(* PLC project mtcs_m2, Institute of Astronomy Onto 0.0.1 *)
(* stored: creationDateTime 2025-03-28T22:57:03.477723, modificationDateTime 2025-03-28T22:57:03.477723 *)

TYPE M2Axes : (X := 0, Y := 1, Z := 2, TILTX := 3, TILTY := 4);
END_TYPE

TYPE M2MoveProcedureStates : (IDLE := 0, ABORTED := 1, PREPARE_PROCESS := 2, MOVING := 3, MOVING_TO_ANTI_BACKLASH_POSITION := 4, MOVING_CLOSE_TO_FINAL_POSITION := 5, MOVING_TO_FINAL_POSITION := 6, ERROR := 7, ABORTING := 8);
END_TYPE

TYPE M2Parts : STRUCT
  {attribute 'TcHmiSymbol.Show'}
  powerRelay : SimpleRelay;  (* Relay to power on/off the power of the M2 field electricity *)
  {attribute 'TcHmiSymbol.Show'}
  heater : SimpleRelay;  (* Digital output to power on/off the heater of M2 *)
  {attribute 'TcHmiSymbol.Show'}
  x : M2XAxis;  (* The X axis *)
  {attribute 'TcHmiSymbol.Show'}
  y : M2YAxis;  (* The Y axis *)
  {attribute 'TcHmiSymbol.Show'}
  z : M2ZAxis;  (* The Z axis *)
  {attribute 'TcHmiSymbol.Show'}
  tiltX : M2TiltXAxis;  (* The TiltX axis *)
  {attribute 'TcHmiSymbol.Show'}
  tiltY : M2TiltYAxis;  (* The TiltY axis *)
  {attribute 'TcHmiSymbol.Show'}
  multiplexer : M2Multiplexer;  (* The multiplexer inputs and outputs *)
  {attribute 'TcHmiSymbol.Show'}
  configManager : ConfigManager;  (* The config manager (to load/save/activate configuration data) *)
  {attribute 'TcHmiSymbol.Show'}
  moveStepsProcedure : M2MoveStepsProcedure;  (* The move steps procedure *)
  {attribute 'TcHmiSymbol.Show'}
  movePositionProcedure : M2MovePositionProcedure;  (* The move to a certain position procedure *)
END_STRUCT;
END_TYPE

TYPE M2MultiplexerParts : STRUCT
  {attribute 'TcHmiSymbol.Show'}
  A : SimpleRelay;  (* Output A of the multiplexer corresponding with the selected axis *)
  {attribute 'TcHmiSymbol.Show'}
  B : SimpleRelay;  (* Output B of the multiplexer corresponding with the selected axis *)
  {attribute 'TcHmiSymbol.Show'}
  C : SimpleRelay;  (* Output C of the multiplexer corresponding with the selected axis *)
  {attribute 'TcHmiSymbol.Show'}
  driveEnable : SimpleRelay;  (* Enabled (TRUE) if the drive selected by the multiplexer must be enabled, Disabled (FALSE) if it must be disabled *)
  {attribute 'TcHmiSymbol.Show'}
  CW : SimpleRelay;  (* Enabled (TRUE) if the motor selected by the multiplexer will run in CW direction (- motion on the screw), Disabled (FALSE) if it will run in CCW direction (+ motion on the screw) *)
  {attribute 'TcHmiSymbol.Show'}
  release : SimpleRelay;  (* Disabled (FALSE) if the motor selected by the multiplexer must be braking, Enabled (TRUE) if it must be released *)
END_STRUCT;
END_TYPE

TYPE M2ZAxisParts : STRUCT
  {attribute 'TcHmiSymbol.Show'}
  highSpeed : SimpleRelay;  (* Enabled (TRUE) to enable the high-speed motion of the Z axis, Disabled (FALSE) to leave it low-speed *)
  {attribute 'TcHmiSymbol.Show'}
  encoder : SSIEncoder;  (* The SSI encoder of the Z axis *)
END_STRUCT;
END_TYPE

TYPE M2Processes : STRUCT
  {attribute 'TcHmiSymbol.Show'}
  initialize : Process;  (* Start initializing *)
  {attribute 'TcHmiSymbol.Show'}
  lock : Process;  (* Lock the system *)
  {attribute 'TcHmiSymbol.Show'}
  unlock : Process;  (* Unlock the system *)
  {attribute 'TcHmiSymbol.Show'}
  changeOperatingState : ChangeOperatingStateProcess;  (* Change the operating state (e.g. AUTO, MANUAL, ...) *)
  {attribute 'TcHmiSymbol.Show'}
  moveAbsolute : M2MoveProcess;  (* Move the position of one axis in an absolute way *)
  {attribute 'TcHmiSymbol.Show'}
  moveRelative : M2MoveProcess;  (* Move the position of one axis relative to the current position *)
  {attribute 'TcHmiSymbol.Show'}
  moveSteps : M2MoveStepsProcess;  (* Move the position of one axis by providing a number of steps (i.e. motor pulses) *)
  {attribute 'TcHmiSymbol.Show'}
  doThermalFocus : Process;  (* Do a thermal focus for the currently active focus *)
  {attribute 'TcHmiSymbol.Show'}
  doThermalFocusForStationName : M2DoThermalFocusForStationName;  (* Do a thermal focus for a specified focal station (based on the configured name of the station) *)
  {attribute 'TcHmiSymbol.Show'}
  doThermalFocusForStationPosition : M2DoThermalFocusForStationPosition;  (* Do a thermal focus for a specified focal station (based on the station numerical ID) *)
  {attribute 'TcHmiSymbol.Show'}
  verifyFixedPositions : Process;  (* Verify (and adjust if necessary) the fixed positions of X, Y, TiltX, and TiltY *)
  {attribute 'TcHmiSymbol.Show'}
  powerOn : Process;  (* Power on the M2 electricity *)
  {attribute 'TcHmiSymbol.Show'}
  powerOff : Process;  (* Power off the M2 electricity *)
  {attribute 'TcHmiSymbol.Show'}
  abort : Process;  (* Abort the move procedure *)
END_STRUCT;
END_TYPE

TYPE M2MultiplexerProcesses : STRUCT
  {attribute 'TcHmiSymbol.Show'}
  selectAxis : M2SelectAxisProcess;  (* Select an axis *)
END_STRUCT;
END_TYPE

TYPE M2Statuses : STRUCT
  {attribute 'TcHmiSymbol.Show'}
  initializationStatus : InitializationStatus;
  {attribute 'TcHmiSymbol.Show'}
  poweredStatus : PoweredStatus;
  {attribute 'TcHmiSymbol.Show'}
  healthStatus : HealthStatus;
  {attribute 'TcHmiSymbol.Show'}
  busyStatus : BusyStatus;
  {attribute 'TcHmiSymbol.Show'}
  operatingStatus : OperatingStatus;
END_STRUCT;
END_TYPE

TYPE M2MultiplexerStatuses : STRUCT
  {attribute 'TcHmiSymbol.Show'}
  healthStatus : HealthStatus;  (* Is the selected drive healthy? *)
  {attribute 'TcHmiSymbol.Show'}
  busyStatus : BusyStatus;  (* Is the selected drive busy? *)
END_STRUCT;
END_TYPE

TYPE M2XAxisStatuses : STRUCT
  {attribute 'TcHmiSymbol.Show'}
  healthStatus : HealthStatus;  (* Is the axis healthy? *)
END_STRUCT;
END_TYPE

TYPE M2YAxisStatuses : STRUCT
  {attribute 'TcHmiSymbol.Show'}
  healthStatus : HealthStatus;  (* Is the axis healthy? *)
END_STRUCT;
END_TYPE

TYPE M2TiltXAxisStatuses : STRUCT
  {attribute 'TcHmiSymbol.Show'}
  healthStatus : HealthStatus;  (* Is the axis healthy? *)
END_STRUCT;
END_TYPE

TYPE M2TiltYAxisStatuses : STRUCT
  {attribute 'TcHmiSymbol.Show'}
  healthStatus : HealthStatus;  (* Is the axis healthy? *)
END_STRUCT;
END_TYPE

TYPE M2ZAxisStatuses : STRUCT
  {attribute 'TcHmiSymbol.Show'}
  healthStatus : HealthStatus;  (* Is the axis healthy? *)
END_STRUCT;
END_TYPE

TYPE M2MoveStepsProcedureStatuses : STRUCT
  {attribute 'TcHmiSymbol.Show'}
  busyStatus : BusyStatus;  (* Is the M2MoveStepsProcedure in a busy state? *)
  {attribute 'TcHmiSymbol.Show'}
  healthStatus : HealthStatus;  (* Is the M2MoveStepsProcedure in a healthy state? *)
END_STRUCT;
END_TYPE

TYPE M2MovePositionProcedureStatuses : STRUCT
  {attribute 'TcHmiSymbol.Show'}
  busyStatus : BusyStatus;  (* Is the M2MoveAbsoluteProcedure in a busy state? *)
  {attribute 'TcHmiSymbol.Show'}
  healthStatus : HealthStatus;  (* Is the M2MoveAbsoluteProcedure in a healthy state? *)
END_STRUCT;
END_TYPE

TYPE M2Config : STRUCT
  {attribute 'TcHmiSymbol.Show'}
  x : M2PotentiometerAxisConfig;  (* The config of the X axis *)
  {attribute 'TcHmiSymbol.Show'}
  y : M2PotentiometerAxisConfig;  (* The config of the Y axis *)
  {attribute 'TcHmiSymbol.Show'}
  z : M2ZAxisConfig;  (* The config of the Z axis *)
  {attribute 'TcHmiSymbol.Show'}
  tiltX : M2PotentiometerAxisConfig;  (* The config of the tiltX axis *)
  {attribute 'TcHmiSymbol.Show'}
  tiltY : M2PotentiometerAxisConfig;  (* The config of the tiltY axis *)
  {attribute 'TcHmiSymbol.Show'}
  thermalFocus : M2ThermalFocusConfig;  (* The thermal focus coefficients for all focal stations *)
  {attribute 'TcHmiSymbol.Show'}
  waitAfterPowerOn : LREAL;  (* Time (in seconds) to wait after the field electricity of M2 have been powered on *)
  {attribute 'TcHmiSymbol.Show'}
  waitAfterPowerOff : LREAL;  (* Time (in seconds) to wait after the field electricity of M2 have been powered off *)
  {attribute 'TcHmiSymbol.Show'}
  powerOffTimeout : LREAL;  (* If no new command is sent to M2 within this time (in seconds) after completion of the last command, M2 will be powered off automatically *)
  {attribute 'TcHmiSymbol.Show'}
  fixedXPosition : LREAL;  (* The fixed X position in mm *)
  {attribute 'TcHmiSymbol.Show'}
  fixedXPositionTolerance : LREAL;  (* If the X position is within fixedXPosition +/- this tolerance, there's no need to adjust it *)
  {attribute 'TcHmiSymbol.Show'}
  fixedYPosition : LREAL;  (* The fixed Y position in mm *)
  {attribute 'TcHmiSymbol.Show'}
  fixedYPositionTolerance : LREAL;  (* If the Y position is within fixedYPosition +/- this tolerance, there's no need to adjust it *)
  {attribute 'TcHmiSymbol.Show'}
  fixedTiltXPosition : LREAL;  (* The fixed TiltX position in mm *)
  {attribute 'TcHmiSymbol.Show'}
  fixedTiltXPositionTolerance : LREAL;  (* If the TiltX position is within fixedTiltXPosition +/- this tolerance, there's no need to adjust it *)
  {attribute 'TcHmiSymbol.Show'}
  fixedTiltYPosition : LREAL;  (* The fixed TiltY position in mm *)
  {attribute 'TcHmiSymbol.Show'}
  fixedTiltYPositionTolerance : LREAL;  (* If the TiltY position is within fixedTiltYPosition +/- this tolerance, there's no need to adjust it *)
  {attribute 'TcHmiSymbol.Show'}
  verifyFixedPositinsOnThermalFocus : BOOL;  (* Each time a theremal focus is done, verify the fixed positions (and adjust them if they fall out of the tolerance) *)
END_STRUCT;
END_TYPE

TYPE M2ThermalFocusStationConfig : STRUCT
  {attribute 'TcHmiSymbol.Show'}
  offset : LREAL;  (* focus = offset + topCoefficient*topTemperature + centreCoefficient*centreTemperature + mirrorCellCoefficient*mirrorCellTemperature *)
  {attribute 'TcHmiSymbol.Show'}
  topCoefficient : LREAL;  (* focus = offset + topCoefficient*topTemperature + centreCoefficient*centreTemperature + mirrorCellCoefficient*mirrorCellTemperature *)
  {attribute 'TcHmiSymbol.Show'}
  centreCoefficient : LREAL;  (* focus = offset + topCoefficient*topTemperature + centreCoefficient*centreTemperature + mirrorCellCoefficient*mirrorCellTemperature *)
  {attribute 'TcHmiSymbol.Show'}
  mirrorCellCoefficient : LREAL;  (* focus = offset + topCoefficient*topTemperature + centreCoefficient*centreTemperature + mirrorCellCoefficient*mirrorCellTemperature *)
END_STRUCT;
END_TYPE

TYPE M2ThermalFocusConfig : STRUCT
  {attribute 'TcHmiSymbol.Show'}
  cassegrain : M2ThermalFocusStationConfig;  (* Cassegrain thermal focus config *)
  {attribute 'TcHmiSymbol.Show'}
  nasmythA : M2ThermalFocusStationConfig;  (* Nasmyth A thermal focus config *)
  {attribute 'TcHmiSymbol.Show'}
  nasmythB : M2ThermalFocusStationConfig;  (* Nasmyth B thermal focus config *)
  {attribute 'TcHmiSymbol.Show'}
  nasmythC : M2ThermalFocusStationConfig;  (* Nasmyth C thermal focus config *)
  {attribute 'TcHmiSymbol.Show'}
  nasmythD : M2ThermalFocusStationConfig;  (* Nasmyth D thermal focus config *)
  {attribute 'TcHmiSymbol.Show'}
  other0 : M2ThermalFocusStationConfig;  (* Other 0 thermal focus config *)
  {attribute 'TcHmiSymbol.Show'}
  other1 : M2ThermalFocusStationConfig;  (* Other 1 thermal focus config *)
  {attribute 'TcHmiSymbol.Show'}
  other2 : M2ThermalFocusStationConfig;  (* Other 2 thermal focus config *)
  {attribute 'TcHmiSymbol.Show'}
  other3 : M2ThermalFocusStationConfig;  (* Other 3 thermal focus config *)
  {attribute 'TcHmiSymbol.Show'}
  other4 : M2ThermalFocusStationConfig;  (* Other 4 thermal focus config *)
END_STRUCT;
END_TYPE

TYPE M2AxisGeneralConfig : STRUCT
  {attribute 'TcHmiSymbol.Show'}
  measurement : MeasurementConfig;  (* Configure the position measurement *)
  {attribute 'TcHmiSymbol.Show'}
  stoppingSteps : UDINT;  (* The number of steps to be expected between the time at which the PLC realizes that the brake release signal must be set, and the time that the axis is fully stopped (for Z axis: at low speed) *)
  {attribute 'TcHmiSymbol.Show'}
  finalSenseCW : BOOL;  (* TRUE if the motor final sense must be ClockWise (- motion on the screw), FALSE if the motor final sense must be CounterClockWise (+ motion on the screw) (for Z axis: at low speed) *)
  {attribute 'TcHmiSymbol.Show'}
  closePosition : UDINT;  (* The number of steps between the Close position (C) and final position (F) *)
  {attribute 'TcHmiSymbol.Show'}
  antiBacklashPosition : UDINT;  (* The number of steps between the Anti-backlash position (A) and final position (F) *)
  {attribute 'TcHmiSymbol.Show'}
  waitAfterMove : LREAL;  (* Time (in seconds) to wait after the axis has been moved *)
  {attribute 'TcHmiSymbol.Show'}
  timeout : LREAL;  (* Timeout for a movement, in seconds (for Z-axis: at low speed) *)
  {attribute 'TcHmiSymbol.Show'}
  verifyPositionOnInitialization : BOOL;  (* Verify the fixed positions (and adjust them if they fall out of the tolerance) during the Initialization procedure *)
END_STRUCT;
END_TYPE

TYPE M2ZAxisConfig : STRUCT
  {attribute 'TcHmiSymbol.Show'}
  general : M2AxisGeneralConfig;  (* Settings which are general for all axes *)
  {attribute 'TcHmiSymbol.Show'}
  highSpeedStoppingSteps : UDINT;  (* The number of steps to be expected between the time at which the PLC realizes that the brake release signal must be set, and the time that the axis is fully stopped at high speed *)
  {attribute 'TcHmiSymbol.Show'}
  highSpeedTimeout : LREAL;  (* Timeout for a fast movement of the Z axis (in seconds) *)
END_STRUCT;
END_TYPE

TYPE M2PotentiometerAxisConfig : STRUCT
  {attribute 'TcHmiSymbol.Show'}
  general : M2AxisGeneralConfig;  (* Settings which are general for all axes *)
  {attribute 'TcHmiSymbol.Show'}
  voltageCorrectionFactor : LREAL;  (* Position = voltage * correctionFactor * voltageToPosition *)
END_STRUCT;
END_TYPE

TYPE M2ConstantsZ : STRUCT
  {attribute 'TcHmiSymbol.Show'}
  MOT_TO_RED_RATIO : LREAL := 134.0;  (* Motor reduction ratio *)
  {attribute 'TcHmiSymbol.Show'}
  RED_TO_SCREW_RATIO : LREAL := 2.0;  (* Transmission ratio between the motor reduction and the screw *)
  {attribute 'TcHmiSymbol.Show'}
  SCREW_TO_ENC_RATIO : LREAL := 1.0;  (* Transmission ratio between the encoder and the screw *)
  {attribute 'TcHmiSymbol.Show'}
  MIN_POSITION : LREAL := 0.0;  (* Minimum position of the axis, in micrometer *)
  {attribute 'TcHmiSymbol.Show'}
  MAX_POSITION : LREAL := 50000.0;  (* Maximum position of the axis, in micrometer *)
  {attribute 'TcHmiSymbol.Show'}
  SCREW_PITCH : LREAL := 2000.0;  (* Screw pitch, in micrometer *)
  {attribute 'TcHmiSymbol.Show'}
  FEEDBACK_RESOLUTION : LREAL := 32.0;  (* Motor feedback resolution (pulses per revolution of the motor rotor) *)
END_STRUCT;
END_TYPE

TYPE M2ConstantsX : STRUCT
  {attribute 'TcHmiSymbol.Show'}
  MOT_TO_RED_RATIO : LREAL := 415.0;  (* Motor reduction ratio *)
  {attribute 'TcHmiSymbol.Show'}
  RED_TO_SCREW_RATIO : LREAL := 2.0;  (* Transmission ratio between the motor reduction and the screw *)
  {attribute 'TcHmiSymbol.Show'}
  SCREW_TO_POT_RATIO : LREAL := 0.5;  (* Transmission ratio between the potentiometer and the screw *)
  {attribute 'TcHmiSymbol.Show'}
  MIN_POSITION : LREAL := 400.0;  (* Minimum position of the axis, in micrometer *)
  {attribute 'TcHmiSymbol.Show'}
  MAX_POSITION : LREAL := 4700.0;  (* Maximum position of the axis, in micrometer *)
  {attribute 'TcHmiSymbol.Show'}
  SCREW_PITCH : LREAL := 1000.0;  (* Screw pitch, in micrometer *)
  {attribute 'TcHmiSymbol.Show'}
  FEEDBACK_RESOLUTION : LREAL := 3.0;  (* Motor feedback resolution (pulses per revolution of the motor rotor) *)
  {attribute 'TcHmiSymbol.Show'}
  POTENTIOMETER_REVOLUTIONS : LREAL := 10.0;  (* Max number of revolutions of the potentiometer *)
END_STRUCT;
END_TYPE

TYPE M2ConstantsY : STRUCT
  {attribute 'TcHmiSymbol.Show'}
  MOT_TO_RED_RATIO : LREAL := 415.0;  (* Motor reduction ratio *)
  {attribute 'TcHmiSymbol.Show'}
  RED_TO_SCREW_RATIO : LREAL := 2.0;  (* Transmission ratio between the motor reduction and the screw *)
  {attribute 'TcHmiSymbol.Show'}
  SCREW_TO_POT_RATIO : LREAL := 0.5;  (* Transmission ratio between the potentiometer and the screw *)
  {attribute 'TcHmiSymbol.Show'}
  MIN_POSITION : LREAL := 400.0;  (* Minimum position of the axis, in micrometer *)
  {attribute 'TcHmiSymbol.Show'}
  MAX_POSITION : LREAL := 4700.0;  (* Maximum position of the axis, in micrometer *)
  {attribute 'TcHmiSymbol.Show'}
  SCREW_PITCH : LREAL := 1000.0;  (* Screw pitch, in micrometer *)
  {attribute 'TcHmiSymbol.Show'}
  FEEDBACK_RESOLUTION : LREAL := 3.0;  (* Motor feedback resolution (pulses per revolution of the motor rotor) *)
  {attribute 'TcHmiSymbol.Show'}
  POTENTIOMETER_REVOLUTIONS : LREAL := 10.0;  (* Max number of revolutions of the potentiometer *)
END_STRUCT;
END_TYPE

TYPE M2ConstantsTiltX : STRUCT
  {attribute 'TcHmiSymbol.Show'}
  MOT_TO_RED_RATIO : LREAL := 1526.0;  (* Motor reduction ratio *)
  {attribute 'TcHmiSymbol.Show'}
  RED_TO_SCREW_RATIO : LREAL := 2.0;  (* Transmission ratio between the motor reduction and the screw *)
  {attribute 'TcHmiSymbol.Show'}
  SCREW_TO_POT_RATIO : LREAL := 0.5;  (* Transmission ratio between the potentiometer and the screw *)
  {attribute 'TcHmiSymbol.Show'}
  MIN_POSITION : LREAL := 260.0;  (* Minimum position of the axis, in micrometer *)
  {attribute 'TcHmiSymbol.Show'}
  MAX_POSITION : LREAL := 1200.0;  (* Maximum position of the axis, in micrometer *)
  {attribute 'TcHmiSymbol.Show'}
  SCREW_PITCH : LREAL := 1000.0;  (* Screw pitch, in micrometer *)
  {attribute 'TcHmiSymbol.Show'}
  FEEDBACK_RESOLUTION : LREAL := 3.0;  (* Motor feedback resolution (pulses per revolution of the motor rotor) *)
  {attribute 'TcHmiSymbol.Show'}
  POTENTIOMETER_REVOLUTIONS : LREAL := 3.0;  (* Max number of revolutions of the potentiometer *)
END_STRUCT;
END_TYPE

TYPE M2ConstantsTiltY : STRUCT
  {attribute 'TcHmiSymbol.Show'}
  MOT_TO_RED_RATIO : LREAL := 1526.0;  (* Motor reduction ratio *)
  {attribute 'TcHmiSymbol.Show'}
  RED_TO_SCREW_RATIO : LREAL := 2.0;  (* Transmission ratio between the motor reduction and the screw *)
  {attribute 'TcHmiSymbol.Show'}
  SCREW_TO_POT_RATIO : LREAL := 0.5;  (* Transmission ratio between the potentiometer and the screw *)
  {attribute 'TcHmiSymbol.Show'}
  MIN_POSITION : LREAL := 180.0;  (* Minimum position of the axis, in micrometer *)
  {attribute 'TcHmiSymbol.Show'}
  MAX_POSITION : LREAL := 1200.0;  (* Maximum position of the axis, in micrometer *)
  {attribute 'TcHmiSymbol.Show'}
  SCREW_PITCH : LREAL := 1000.0;  (* Screw pitch, in micrometer *)
  {attribute 'TcHmiSymbol.Show'}
  FEEDBACK_RESOLUTION : LREAL := 3.0;  (* Motor feedback resolution (pulses per revolution of the motor rotor) *)
  {attribute 'TcHmiSymbol.Show'}
  POTENTIOMETER_REVOLUTIONS : LREAL := 3.0;  (* Max number of revolutions of the potentiometer *)
END_STRUCT;
END_TYPE

TYPE M2SelectAxisProcessArgs : STRUCT
  {attribute 'TcHmiSymbol.Show'}
  axis : M2Axes;  (* The axis to select *)
END_STRUCT;
END_TYPE

TYPE M2MoveProcessArgs : STRUCT
  {attribute 'TcHmiSymbol.Show'}
  axis : M2Axes;  (* The axis to move *)
  {attribute 'TcHmiSymbol.Show'}
  position : LREAL;  (* Move to a certain position in millimeters *)
END_STRUCT;
END_TYPE

TYPE M2MoveStepsProcessArgs : STRUCT
  {attribute 'TcHmiSymbol.Show'}
  axis : M2Axes;  (* The axis to move *)
  {attribute 'TcHmiSymbol.Show'}
  steps : UDINT;  (* Move a certain number of steps *)
  {attribute 'TcHmiSymbol.Show'}
  cw : BOOL;  (* True if the axis should be moved in CW (negative) direction *)
  {attribute 'TcHmiSymbol.Show'}
  fast : BOOL;  (* True if the axis should be moved fast (only used in case of Z-axis!) *)
END_STRUCT;
END_TYPE

TYPE M2DoThermalFocusForStationPositionArgs : STRUCT
  {attribute 'TcHmiSymbol.Show'}
  station : M3PositionIDs;  (* The station numerical ID for which the thermal focus should be executed *)
END_STRUCT;
END_TYPE

TYPE M2DoThermalFocusForStationNameArgs : STRUCT
  {attribute 'TcHmiSymbol.Show'}
  station : STRING;  (* The configured station name, for which the thermal focus should be executed *)
END_STRUCT;
END_TYPE

FUNCTION_BLOCK SM_M2
  VAR_INPUT
    {attribute 'TcHmiSymbol.Show'}
    {attribute 'OPC.UA.DA' := '1'}
    {attribute 'OPC.UA.DA.Access' := '1'}
    editableConfig : M2Config;  (* Editable configuration of the M2 subsystem *)
  END_VAR
  VAR_OUTPUT
    {attribute 'OPC.UA.DA' := '1'}
    {attribute 'OPC.UA.DA.Access' := '1'}
    {attribute 'TcHmiSymbol.Show'}
    actualStatus : STRING;  (* Current status description *)
    {attribute 'TcHmiSymbol.Show'}
    previousStatus : STRING;  (* Previous status description *)
    {attribute 'TcHmiSymbol.Show'}
    {attribute 'OPC.UA.DA' := '1'}
    {attribute 'OPC.UA.DA.Access' := '1'}
    config : M2Config;  (* Active configuration of the M2 subsystem *)
    {attribute 'TcHmiSymbol.Show'}
    {attribute 'OPC.UA.DA' := '1'}
    {attribute 'OPC.UA.DA.Access' := '1'}
    selectedAxis : M2Axes;  (* The axis which is currently selected by the multiplexer *)
    {attribute 'TcHmiSymbol.Show'}
    {attribute 'OPC.UA.DA' := '1'}
    {attribute 'OPC.UA.DA.Access' := '1'}
    selectedAxisName : STRING;  (* The name of the axis which is currently selected by the multiplexer *)
    {attribute 'TcHmiSymbol.Show'}
    {attribute 'OPC.UA.DA' := '1'}
    {attribute 'OPC.UA.DA.Access' := '1'}
    powerOffTimer : LREAL;  (* Number of seconds before the power of the M2 field electricity will be powered off automatically *)
    {attribute 'TcHmiSymbol.Show'}
    {attribute 'OPC.UA.DA' := '1'}
    {attribute 'OPC.UA.DA.Access' := '1'}
    thermalFocusCassegrain : LinearPosition;  (* Thermal focus position for cassegrain *)
    {attribute 'TcHmiSymbol.Show'}
    {attribute 'OPC.UA.DA' := '1'}
    {attribute 'OPC.UA.DA.Access' := '1'}
    thermalFocusNasmythA : LinearPosition;  (* Thermal focus position for nasmyth A *)
    {attribute 'TcHmiSymbol.Show'}
    {attribute 'OPC.UA.DA' := '1'}
    {attribute 'OPC.UA.DA.Access' := '1'}
    thermalFocusNasmythB : LinearPosition;  (* Thermal focus position for nasmyth B *)
    {attribute 'TcHmiSymbol.Show'}
    {attribute 'OPC.UA.DA' := '1'}
    {attribute 'OPC.UA.DA.Access' := '1'}
    thermalFocusNasmythC : LinearPosition;  (* Thermal focus position for nasmyth C *)
    {attribute 'TcHmiSymbol.Show'}
    {attribute 'OPC.UA.DA' := '1'}
    {attribute 'OPC.UA.DA.Access' := '1'}
    thermalFocusNasmythD : LinearPosition;  (* Thermal focus position for nasmyth D *)
    {attribute 'TcHmiSymbol.Show'}
    {attribute 'OPC.UA.DA' := '1'}
    {attribute 'OPC.UA.DA.Access' := '1'}
    thermalFocusActualFocalStation : LinearPosition;  (* Thermal focus position for nasmyth D *)
    {attribute 'TcHmiSymbol.Show'}
    statuses : M2Statuses;  (* Statuses of the state machine *)
    {attribute 'TcHmiSymbol.Show'}
    parts : M2Parts;  (* Parts of the state machine *)
    {attribute 'TcHmiSymbol.Show'}
    processes : M2Processes;  (* Processes of the state machine *)
  END_VAR
  VAR_IN_OUT
    {attribute 'TcHmiSymbol.Show'}
    {attribute 'OPC.UA.DA' := '0'}
    {attribute 'TcHmiSymbol.Hide'}
    operatorStatus : OperatorStatus;  (* Shared operator status *)
    {attribute 'TcHmiSymbol.Show'}
    {attribute 'OPC.UA.DA' := '0'}
    {attribute 'TcHmiSymbol.Hide'}
    io : M1M2IO;  (* Shared I/O with M1 *)
    {attribute 'TcHmiSymbol.Show'}
    {attribute 'OPC.UA.DA' := '0'}
    {attribute 'TcHmiSymbol.Hide'}
    actualFocalStation : M3PositionIDs;  (* Actual M3 focal station, needed for thermal focus *)
    {attribute 'TcHmiSymbol.Show'}
    {attribute 'OPC.UA.DA' := '0'}
    {attribute 'TcHmiSymbol.Hide'}
    m3KnownPositionsConfig : M3KnownPositionsConfig;  (* Config of M3 with all info (e.g. names) of focal stations *)
    {attribute 'TcHmiSymbol.Show'}
    {attribute 'OPC.UA.DA' := '0'}
    {attribute 'TcHmiSymbol.Hide'}
    temperatures : TelemetryTemperatures;  (* Telemetry temperatures *)
  END_VAR

            parts.powerRelay( isEnabled := operatorStatus.tech );
parts.heater( isEnabled := operatorStatus.tech );
parts.x(
    powered := statuses.poweredStatus.enabled,
    config := config,
    axisConfig := config.x);
parts.y(
    powered := statuses.poweredStatus.enabled,
    config := config,
    axisConfig := config.y);
parts.z(
    powered := statuses.poweredStatus.enabled,
    config := config,
    axisConfig := config.z,
    isEnabled := operatorStatus.tech);
parts.tiltX(
    powered := statuses.poweredStatus.enabled,
    config := config,
    axisConfig := config.tiltX);
parts.tiltY(
    powered := statuses.poweredStatus.enabled,
    config := config,
    axisConfig := config.tiltY);
parts.multiplexer(
    isEnabled := operatorStatus.tech,
    powered := statuses.poweredStatus.enabled);
parts.configManager( isEnabled := operatorStatus.tech );
parts.moveStepsProcedure(
    powerOn := processes.powerOn,
    x := parts.x,
    y := parts.y,
    z := parts.z,
    tiltX := parts.tiltX,
    tiltY := parts.tiltY,
    multiplexer := parts.multiplexer,
    config := config);
parts.movePositionProcedure(
    powerOn := processes.powerOn,
    x := parts.x,
    y := parts.y,
    z := parts.z,
    tiltX := parts.tiltX,
    tiltY := parts.tiltY,
    multiplexer := parts.multiplexer,
    moveStepsProcedure := parts.moveStepsProcedure,
    config := config);
statuses.initializationStatus();
statuses.poweredStatus( isEnabled := parts.powerRelay.digitalOutput AND (processes.powerOn.statuses.busyStatus.idle AND processes.powerOff.statuses.busyStatus.idle) );
statuses.healthStatus(
    isGood := ((parts.x.statuses.healthStatus.isGood AND (parts.y.statuses.healthStatus.isGood AND (parts.z.statuses.healthStatus.isGood AND (parts.tiltX.statuses.healthStatus.isGood AND (parts.tiltY.statuses.healthStatus.isGood AND parts.multiplexer.statuses.healthStatus.isGood))))) OR statuses.poweredStatus.disabled) AND (io.statuses.healthStatus.isGood AND (temperatures.statuses.healthStatus.isGood AND parts.configManager.statuses.healthStatus.isGood)),
    hasWarning := ((parts.x.statuses.healthStatus.hasWarning OR (parts.y.statuses.healthStatus.hasWarning OR (parts.z.statuses.healthStatus.hasWarning OR (parts.tiltX.statuses.healthStatus.hasWarning OR (parts.tiltY.statuses.healthStatus.hasWarning OR parts.multiplexer.statuses.healthStatus.hasWarning))))) AND statuses.poweredStatus.enabled) OR (io.statuses.healthStatus.hasWarning OR (temperatures.statuses.healthStatus.hasWarning OR parts.configManager.statuses.healthStatus.hasWarning)));
statuses.busyStatus( isBusy := statuses.initializationStatus.initializing OR (parts.multiplexer.statuses.busyStatus.busy OR (parts.configManager.statuses.busyStatus.busy OR (processes.abort.statuses.busyStatus.busy OR (processes.powerOn.statuses.busyStatus.busy OR (processes.powerOff.statuses.busyStatus.busy OR (processes.doThermalFocus.statuses.busyStatus.busy OR (processes.doThermalFocusForStationName.statuses.busyStatus.busy OR (processes.doThermalFocusForStationPosition.statuses.busyStatus.busy OR (processes.verifyFixedPositions.statuses.busyStatus.busy OR (processes.moveSteps.statuses.busyStatus.busy OR (processes.moveAbsolute.statuses.busyStatus.busy OR processes.moveRelative.statuses.busyStatus.busy))))))))))) );
statuses.operatingStatus( superState := statuses.initializationStatus.initialized );
processes.initialize( isEnabled := statuses.initializationStatus.shutdown OR (statuses.initializationStatus.initializingFailed OR statuses.initializationStatus.initialized) );
processes.lock( isEnabled := operatorStatus.tech AND statuses.initializationStatus.initialized );
processes.unlock( isEnabled := operatorStatus.tech AND statuses.initializationStatus.locked );
processes.changeOperatingState( isEnabled := statuses.busyStatus.idle AND (statuses.initializationStatus.initialized AND operatorStatus.tech) );
processes.moveAbsolute( isEnabled := statuses.initializationStatus.initialized AND statuses.busyStatus.idle );
processes.moveRelative( isEnabled := processes.moveAbsolute.isEnabled );
processes.moveSteps( isEnabled := statuses.initializationStatus.initialized AND operatorStatus.tech );
processes.doThermalFocus( isEnabled := processes.moveAbsolute.isEnabled AND (NOT(actualFocalStation = M3PositionIDs.UNKNOWN)) );
processes.doThermalFocusForStationName( isEnabled := processes.moveAbsolute.isEnabled );
processes.doThermalFocusForStationPosition( isEnabled := processes.moveAbsolute.isEnabled );
processes.verifyFixedPositions( isEnabled := processes.moveAbsolute.isEnabled );
processes.powerOn( isEnabled := statuses.busyStatus.idle AND statuses.initializationStatus.initialized );
processes.powerOff( isEnabled := statuses.busyStatus.idle AND statuses.initializationStatus.initialized );
processes.abort( isEnabled := parts.moveStepsProcedure.statuses.busyStatus.busy OR parts.movePositionProcedure.statuses.busyStatus.busy );

          

{attribute 'TcRpcEnable' := '1'}
METHOD initialize : RequestResults
                  initialize := THIS^.processes.initialize.request();

                
END_METHOD

{attribute 'TcRpcEnable' := '1'}
METHOD lock : RequestResults
                  lock := THIS^.processes.lock.request();

                
END_METHOD

{attribute 'TcRpcEnable' := '1'}
METHOD unlock : RequestResults
                  unlock := THIS^.processes.unlock.request();

                
END_METHOD

{attribute 'TcRpcEnable' := '1'}
METHOD changeOperatingState : RequestResults
  VAR_INPUT
    {attribute 'TcHmiSymbol.Show'}
    state : OperatingStates;
  END_VAR
                  changeOperatingState := THIS^.processes.changeOperatingState.request( state := state );

                
END_METHOD

{attribute 'TcRpcEnable' := '1'}
METHOD moveAbsolute : RequestResults
  VAR_INPUT
    {attribute 'TcHmiSymbol.Show'}
    axis : M2Axes;
    {attribute 'TcHmiSymbol.Show'}
    position : LREAL;
  END_VAR
                  moveAbsolute := THIS^.processes.moveAbsolute.request(
    axis := axis,
    position := position);

                
END_METHOD

{attribute 'TcRpcEnable' := '1'}
METHOD moveRelative : RequestResults
  VAR_INPUT
    {attribute 'TcHmiSymbol.Show'}
    axis : M2Axes;
    {attribute 'TcHmiSymbol.Show'}
    position : LREAL;
  END_VAR
                  moveRelative := THIS^.processes.moveRelative.request(
    axis := axis,
    position := position);

                
END_METHOD

{attribute 'TcRpcEnable' := '1'}
METHOD moveSteps : RequestResults
  VAR_INPUT
    {attribute 'TcHmiSymbol.Show'}
    axis : M2Axes;
    {attribute 'TcHmiSymbol.Show'}
    steps : UDINT;
    {attribute 'TcHmiSymbol.Show'}
    cw : BOOL;
    {attribute 'TcHmiSymbol.Show'}
    fast : BOOL;
  END_VAR
                  moveSteps := THIS^.processes.moveSteps.request(
    axis := axis,
    steps := steps,
    cw := cw,
    fast := fast);

                
END_METHOD

{attribute 'TcRpcEnable' := '1'}
METHOD doThermalFocus : RequestResults
                  doThermalFocus := THIS^.processes.doThermalFocus.request();

                
END_METHOD

{attribute 'TcRpcEnable' := '1'}
METHOD doThermalFocusForStationName : RequestResults
  VAR_INPUT
    {attribute 'TcHmiSymbol.Show'}
    station : STRING;
  END_VAR
                  doThermalFocusForStationName := THIS^.processes.doThermalFocusForStationName.request( station := station );

                
END_METHOD

{attribute 'TcRpcEnable' := '1'}
METHOD doThermalFocusForStationPosition : RequestResults
  VAR_INPUT
    {attribute 'TcHmiSymbol.Show'}
    station : M3PositionIDs;
  END_VAR
                  doThermalFocusForStationPosition := THIS^.processes.doThermalFocusForStationPosition.request( station := station );

                
END_METHOD

{attribute 'TcRpcEnable' := '1'}
METHOD verifyFixedPositions : RequestResults
                  verifyFixedPositions := THIS^.processes.verifyFixedPositions.request();

                
END_METHOD

{attribute 'TcRpcEnable' := '1'}
METHOD powerOn : RequestResults
                  powerOn := THIS^.processes.powerOn.request();

                
END_METHOD

{attribute 'TcRpcEnable' := '1'}
METHOD powerOff : RequestResults
                  powerOff := THIS^.processes.powerOff.request();

                
END_METHOD

{attribute 'TcRpcEnable' := '1'}
METHOD abort : RequestResults
                  abort := THIS^.processes.abort.request();

                
END_METHOD

METHOD _log : BOOL
  VAR_INPUT
    {attribute 'TcHmiSymbol.Show'}
    name : STRING;  (* Name of this function block instance *)
  END_VAR
  VAR_IN_OUT
    {attribute 'TcHmiSymbol.Show'}
    buffer : LogBuffer;  (* Buffer to write all logging to *)
  END_VAR
  VAR
    {attribute 'TcHmiSymbol.Show'}
    subBuffer : LogBuffer;  (* Temporary buffer to write logging by parts (sub-statemachines) to *)
  END_VAR
                  THIS^.parts.powerRelay._log(
    name := 'powerRelay',
    buffer := subBuffer);
THIS^.parts.heater._log(
    name := 'heater',
    buffer := subBuffer);
THIS^.parts.x._log(
    name := 'x',
    buffer := subBuffer);
THIS^.parts.y._log(
    name := 'y',
    buffer := subBuffer);
THIS^.parts.z._log(
    name := 'z',
    buffer := subBuffer);
THIS^.parts.tiltX._log(
    name := 'tiltX',
    buffer := subBuffer);
THIS^.parts.tiltY._log(
    name := 'tiltY',
    buffer := subBuffer);
THIS^.parts.multiplexer._log(
    name := 'multiplexer',
    buffer := subBuffer);
THIS^.parts.configManager._log(
    name := 'configManager',
    buffer := subBuffer);
THIS^.parts.moveStepsProcedure._log(
    name := 'moveStepsProcedure',
    buffer := subBuffer);
THIS^.parts.movePositionProcedure._log(
    name := 'movePositionProcedure',
    buffer := subBuffer);
THIS^.processes.initialize._log(
    name := 'processes.initialize',
    buffer := subBuffer);
THIS^.processes.lock._log(
    name := 'processes.lock',
    buffer := subBuffer);
THIS^.processes.unlock._log(
    name := 'processes.unlock',
    buffer := subBuffer);
THIS^.processes.changeOperatingState._log(
    name := 'processes.changeOperatingState',
    buffer := subBuffer);
THIS^.processes.moveAbsolute._log(
    name := 'processes.moveAbsolute',
    buffer := subBuffer);
THIS^.processes.moveRelative._log(
    name := 'processes.moveRelative',
    buffer := subBuffer);
THIS^.processes.moveSteps._log(
    name := 'processes.moveSteps',
    buffer := subBuffer);
THIS^.processes.doThermalFocus._log(
    name := 'processes.doThermalFocus',
    buffer := subBuffer);
THIS^.processes.doThermalFocusForStationName._log(
    name := 'processes.doThermalFocusForStationName',
    buffer := subBuffer);
THIS^.processes.doThermalFocusForStationPosition._log(
    name := 'processes.doThermalFocusForStationPosition',
    buffer := subBuffer);
THIS^.processes.verifyFixedPositions._log(
    name := 'processes.verifyFixedPositions',
    buffer := subBuffer);
THIS^.processes.powerOn._log(
    name := 'processes.powerOn',
    buffer := subBuffer);
THIS^.processes.powerOff._log(
    name := 'processes.powerOff',
    buffer := subBuffer);
THIS^.processes.abort._log(
    name := 'processes.abort',
    buffer := subBuffer);
LOGGER(
    name := name,
    actualStatus := THIS^.actualStatus,
    previousStatus := THIS^.previousStatus,
    buffer := buffer,
    subBuffer := subBuffer,
    pHealthStatus := ADR(THIS^.statuses.healthStatus),
    pBusyStatus := ADR(THIS^.statuses.busyStatus));

                
END_METHOD
END_FUNCTION_BLOCK

FUNCTION_BLOCK SM_M2Multiplexer
  VAR_INPUT
    {attribute 'TcHmiSymbol.Show'}
    {attribute 'OPC.UA.DA' := '1'}
    {attribute 'OPC.UA.DA.Access' := '1'}
    noFault AT %I* : BOOL;  (* FALSE if the drive selected by the multiplexer is in faulty state, TRUE if it is in a healthy state *)
    {attribute 'TcHmiSymbol.Show'}
    {attribute 'OPC.UA.DA' := '1'}
    {attribute 'OPC.UA.DA.Access' := '1'}
    isEnabled : BOOL;  (* TRUE if the multiplexer is enabled, FALSE if not *)
    {attribute 'TcHmiSymbol.Show'}
    {attribute 'OPC.UA.DA' := '1'}
    {attribute 'OPC.UA.DA.Access' := '1'}
    powered : BOOL;  (* TRUE if the axis is powered *)
  END_VAR
  VAR_OUTPUT
    {attribute 'OPC.UA.DA' := '1'}
    {attribute 'OPC.UA.DA.Access' := '1'}
    {attribute 'TcHmiSymbol.Show'}
    actualStatus : STRING;  (* Current status description *)
    {attribute 'TcHmiSymbol.Show'}
    previousStatus : STRING;  (* Previous status description *)
    {attribute 'TcHmiSymbol.Show'}
    statuses : M2MultiplexerStatuses;  (* Statuses of the state machine *)
    {attribute 'TcHmiSymbol.Show'}
    parts : M2MultiplexerParts;  (* Parts of the state machine *)
    {attribute 'TcHmiSymbol.Show'}
    processes : M2MultiplexerProcesses;  (* Processes of the state machine *)
  END_VAR
  VAR
    {attribute 'TcHmiSymbol.Show'}
    {attribute 'OPC.UA.DA' := '1'}
    {attribute 'OPC.UA.DA.Access' := '1'}
    noFault_ro : BOOL;
  END_VAR

            parts.A( isEnabled := isEnabled );
parts.B( isEnabled := isEnabled );
parts.C( isEnabled := isEnabled );
parts.driveEnable( isEnabled := isEnabled );
parts.CW( isEnabled := isEnabled );
parts.release( isEnabled := isEnabled );
statuses.healthStatus( isGood := (noFault OR (NOT(powered))) AND processes.selectAxis.statuses.healthStatus.good );
statuses.busyStatus( isBusy := parts.A.statuses.busyStatus.busy OR (parts.B.statuses.busyStatus.busy OR (parts.C.statuses.busyStatus.busy OR (parts.driveEnable.statuses.busyStatus.busy OR (parts.CW.statuses.busyStatus.busy OR parts.release.statuses.busyStatus.busy)))) );
processes.selectAxis( isEnabled := isEnabled );
noFault_ro := noFault;

          

{attribute 'TcRpcEnable' := '1'}
METHOD selectAxis : RequestResults
  VAR_INPUT
    {attribute 'TcHmiSymbol.Show'}
    axis : M2Axes;
  END_VAR
                  selectAxis := THIS^.processes.selectAxis.request( axis := axis );

                
END_METHOD

METHOD _log : BOOL
  VAR_INPUT
    {attribute 'TcHmiSymbol.Show'}
    name : STRING;  (* Name of this function block instance *)
  END_VAR
  VAR_IN_OUT
    {attribute 'TcHmiSymbol.Show'}
    buffer : LogBuffer;  (* Buffer to write all logging to *)
  END_VAR
  VAR
    {attribute 'TcHmiSymbol.Show'}
    subBuffer : LogBuffer;  (* Temporary buffer to write logging by parts (sub-statemachines) to *)
  END_VAR
                  THIS^.parts.A._log(
    name := 'A',
    buffer := subBuffer);
THIS^.parts.B._log(
    name := 'B',
    buffer := subBuffer);
THIS^.parts.C._log(
    name := 'C',
    buffer := subBuffer);
THIS^.parts.driveEnable._log(
    name := 'driveEnable',
    buffer := subBuffer);
THIS^.parts.CW._log(
    name := 'CW',
    buffer := subBuffer);
THIS^.parts.release._log(
    name := 'release',
    buffer := subBuffer);
THIS^.processes.selectAxis._log(
    name := 'processes.selectAxis',
    buffer := subBuffer);
LOGGER(
    name := name,
    actualStatus := THIS^.actualStatus,
    previousStatus := THIS^.previousStatus,
    buffer := buffer,
    subBuffer := subBuffer,
    pHealthStatus := ADR(THIS^.statuses.healthStatus),
    pBusyStatus := ADR(THIS^.statuses.busyStatus));

                
END_METHOD
END_FUNCTION_BLOCK

FUNCTION_BLOCK SM_M2XAxis
  VAR_INPUT
    {attribute 'TcHmiSymbol.Show'}
    {attribute 'OPC.UA.DA' := '1'}
    {attribute 'OPC.UA.DA.Access' := '1'}
    position : LinearPositionMeasurement16;  (* Actual position of the axis *)
    {attribute 'TcHmiSymbol.Show'}
    {attribute 'OPC.UA.DA' := '1'}
    {attribute 'OPC.UA.DA.Access' := '1'}
    backlashLifted : BOOL;  (* TRUE if the backlash was previously lifted *)
    {attribute 'TcHmiSymbol.Show'}
    {attribute 'OPC.UA.DA' := '1'}
    {attribute 'OPC.UA.DA.Access' := '1'}
    powered : BOOL;  (* TRUE if the axis is powered *)
  END_VAR
  VAR_OUTPUT
    {attribute 'OPC.UA.DA' := '1'}
    {attribute 'OPC.UA.DA.Access' := '1'}
    {attribute 'TcHmiSymbol.Show'}
    actualStatus : STRING;  (* Current status description *)
    {attribute 'TcHmiSymbol.Show'}
    previousStatus : STRING;  (* Previous status description *)
    {attribute 'TcHmiSymbol.Show'}
    {attribute 'OPC.UA.DA' := '1'}
    {attribute 'OPC.UA.DA.Access' := '1'}
    constants : M2ConstantsX;  (* Some constants particular for this axis *)
    {attribute 'TcHmiSymbol.Show'}
    statuses : M2XAxisStatuses;  (* Statuses of the state machine *)
  END_VAR
  VAR_IN_OUT
    {attribute 'TcHmiSymbol.Show'}
    {attribute 'OPC.UA.DA' := '0'}
    {attribute 'TcHmiSymbol.Hide'}
    config : M2Config;  (* The general M2 config *)
    {attribute 'TcHmiSymbol.Show'}
    {attribute 'OPC.UA.DA' := '0'}
    {attribute 'TcHmiSymbol.Hide'}
    axisConfig : M2PotentiometerAxisConfig;  (* The config particular for this axis *)
  END_VAR

            position(
    config := axisConfig.general.measurement,
    conversionFactor := (constants.POTENTIOMETER_REVOLUTIONS * (constants.SCREW_TO_POT_RATIO * constants.SCREW_PITCH)) / (32768.0 * 1000.0));
statuses.healthStatus(
    isGood := position.statuses.healthStatus.isGood,
    hasWarning := position.statuses.healthStatus.hasWarning);

          

METHOD _log : BOOL
  VAR_INPUT
    {attribute 'TcHmiSymbol.Show'}
    name : STRING;  (* Name of this function block instance *)
  END_VAR
  VAR_IN_OUT
    {attribute 'TcHmiSymbol.Show'}
    buffer : LogBuffer;  (* Buffer to write all logging to *)
  END_VAR
  VAR
    {attribute 'TcHmiSymbol.Show'}
    subBuffer : LogBuffer;  (* Temporary buffer to write logging by parts (sub-statemachines) to *)
  END_VAR
                  LOGGER(
    name := name,
    actualStatus := THIS^.actualStatus,
    previousStatus := THIS^.previousStatus,
    buffer := buffer,
    subBuffer := subBuffer,
    pHealthStatus := ADR(THIS^.statuses.healthStatus));

                
END_METHOD
END_FUNCTION_BLOCK

FUNCTION_BLOCK SM_M2YAxis
  VAR_INPUT
    {attribute 'TcHmiSymbol.Show'}
    {attribute 'OPC.UA.DA' := '1'}
    {attribute 'OPC.UA.DA.Access' := '1'}
    position : LinearPositionMeasurement16;  (* Actual position of the axis *)
    {attribute 'TcHmiSymbol.Show'}
    {attribute 'OPC.UA.DA' := '1'}
    {attribute 'OPC.UA.DA.Access' := '1'}
    backlashLifted : BOOL;  (* TRUE if the backlash was previously lifted *)
    {attribute 'TcHmiSymbol.Show'}
    {attribute 'OPC.UA.DA' := '1'}
    {attribute 'OPC.UA.DA.Access' := '1'}
    powered : BOOL;  (* TRUE if the axis is powered *)
  END_VAR
  VAR_OUTPUT
    {attribute 'OPC.UA.DA' := '1'}
    {attribute 'OPC.UA.DA.Access' := '1'}
    {attribute 'TcHmiSymbol.Show'}
    actualStatus : STRING;  (* Current status description *)
    {attribute 'TcHmiSymbol.Show'}
    previousStatus : STRING;  (* Previous status description *)
    {attribute 'TcHmiSymbol.Show'}
    {attribute 'OPC.UA.DA' := '1'}
    {attribute 'OPC.UA.DA.Access' := '1'}
    constants : M2ConstantsY;  (* Some constants particular for this axis *)
    {attribute 'TcHmiSymbol.Show'}
    statuses : M2YAxisStatuses;  (* Statuses of the state machine *)
  END_VAR
  VAR_IN_OUT
    {attribute 'TcHmiSymbol.Show'}
    {attribute 'OPC.UA.DA' := '0'}
    {attribute 'TcHmiSymbol.Hide'}
    config : M2Config;  (* The general M2 config *)
    {attribute 'TcHmiSymbol.Show'}
    {attribute 'OPC.UA.DA' := '0'}
    {attribute 'TcHmiSymbol.Hide'}
    axisConfig : M2PotentiometerAxisConfig;  (* The config particular for this axis *)
  END_VAR

            position(
    config := axisConfig.general.measurement,
    conversionFactor := (constants.POTENTIOMETER_REVOLUTIONS * (constants.SCREW_TO_POT_RATIO * constants.SCREW_PITCH)) / (32768.0 * 1000.0));
statuses.healthStatus(
    isGood := position.statuses.healthStatus.isGood,
    hasWarning := position.statuses.healthStatus.hasWarning);

          

METHOD _log : BOOL
  VAR_INPUT
    {attribute 'TcHmiSymbol.Show'}
    name : STRING;  (* Name of this function block instance *)
  END_VAR
  VAR_IN_OUT
    {attribute 'TcHmiSymbol.Show'}
    buffer : LogBuffer;  (* Buffer to write all logging to *)
  END_VAR
  VAR
    {attribute 'TcHmiSymbol.Show'}
    subBuffer : LogBuffer;  (* Temporary buffer to write logging by parts (sub-statemachines) to *)
  END_VAR
                  LOGGER(
    name := name,
    actualStatus := THIS^.actualStatus,
    previousStatus := THIS^.previousStatus,
    buffer := buffer,
    subBuffer := subBuffer,
    pHealthStatus := ADR(THIS^.statuses.healthStatus));

                
END_METHOD
END_FUNCTION_BLOCK

FUNCTION_BLOCK SM_M2TiltXAxis
  VAR_INPUT
    {attribute 'TcHmiSymbol.Show'}
    {attribute 'OPC.UA.DA' := '1'}
    {attribute 'OPC.UA.DA.Access' := '1'}
    position : LinearPositionMeasurement16;  (* Actual position of the axis *)
    {attribute 'TcHmiSymbol.Show'}
    {attribute 'OPC.UA.DA' := '1'}
    {attribute 'OPC.UA.DA.Access' := '1'}
    backlashLifted : BOOL;  (* TRUE if the backlash was previously lifted *)
    {attribute 'TcHmiSymbol.Show'}
    {attribute 'OPC.UA.DA' := '1'}
    {attribute 'OPC.UA.DA.Access' := '1'}
    powered : BOOL;  (* TRUE if the axis is powered *)
  END_VAR
  VAR_OUTPUT
    {attribute 'OPC.UA.DA' := '1'}
    {attribute 'OPC.UA.DA.Access' := '1'}
    {attribute 'TcHmiSymbol.Show'}
    actualStatus : STRING;  (* Current status description *)
    {attribute 'TcHmiSymbol.Show'}
    previousStatus : STRING;  (* Previous status description *)
    {attribute 'TcHmiSymbol.Show'}
    {attribute 'OPC.UA.DA' := '1'}
    {attribute 'OPC.UA.DA.Access' := '1'}
    constants : M2ConstantsTiltX;  (* Some constants particular for this axis *)
    {attribute 'TcHmiSymbol.Show'}
    statuses : M2TiltXAxisStatuses;  (* Statuses of the state machine *)
  END_VAR
  VAR_IN_OUT
    {attribute 'TcHmiSymbol.Show'}
    {attribute 'OPC.UA.DA' := '0'}
    {attribute 'TcHmiSymbol.Hide'}
    config : M2Config;  (* The general M2 config *)
    {attribute 'TcHmiSymbol.Show'}
    {attribute 'OPC.UA.DA' := '0'}
    {attribute 'TcHmiSymbol.Hide'}
    axisConfig : M2PotentiometerAxisConfig;  (* The config particular for this axis *)
  END_VAR

            position(
    config := axisConfig.general.measurement,
    conversionFactor := (constants.POTENTIOMETER_REVOLUTIONS * (constants.SCREW_TO_POT_RATIO * constants.SCREW_PITCH)) / (32768.0 * 1000.0));
statuses.healthStatus(
    isGood := position.statuses.healthStatus.isGood,
    hasWarning := position.statuses.healthStatus.hasWarning);

          

METHOD _log : BOOL
  VAR_INPUT
    {attribute 'TcHmiSymbol.Show'}
    name : STRING;  (* Name of this function block instance *)
  END_VAR
  VAR_IN_OUT
    {attribute 'TcHmiSymbol.Show'}
    buffer : LogBuffer;  (* Buffer to write all logging to *)
  END_VAR
  VAR
    {attribute 'TcHmiSymbol.Show'}
    subBuffer : LogBuffer;  (* Temporary buffer to write logging by parts (sub-statemachines) to *)
  END_VAR
                  LOGGER(
    name := name,
    actualStatus := THIS^.actualStatus,
    previousStatus := THIS^.previousStatus,
    buffer := buffer,
    subBuffer := subBuffer,
    pHealthStatus := ADR(THIS^.statuses.healthStatus));

                
END_METHOD
END_FUNCTION_BLOCK

FUNCTION_BLOCK SM_M2TiltYAxis
  VAR_INPUT
    {attribute 'TcHmiSymbol.Show'}
    {attribute 'OPC.UA.DA' := '1'}
    {attribute 'OPC.UA.DA.Access' := '1'}
    position : LinearPositionMeasurement16;  (* Actual position of the axis *)
    {attribute 'TcHmiSymbol.Show'}
    {attribute 'OPC.UA.DA' := '1'}
    {attribute 'OPC.UA.DA.Access' := '1'}
    backlashLifted : BOOL;  (* TRUE if the backlash was previously lifted *)
    {attribute 'TcHmiSymbol.Show'}
    {attribute 'OPC.UA.DA' := '1'}
    {attribute 'OPC.UA.DA.Access' := '1'}
    powered : BOOL;  (* TRUE if the axis is powered *)
  END_VAR
  VAR_OUTPUT
    {attribute 'OPC.UA.DA' := '1'}
    {attribute 'OPC.UA.DA.Access' := '1'}
    {attribute 'TcHmiSymbol.Show'}
    actualStatus : STRING;  (* Current status description *)
    {attribute 'TcHmiSymbol.Show'}
    previousStatus : STRING;  (* Previous status description *)
    {attribute 'TcHmiSymbol.Show'}
    {attribute 'OPC.UA.DA' := '1'}
    {attribute 'OPC.UA.DA.Access' := '1'}
    constants : M2ConstantsTiltY;  (* Some constants particular for this axis *)
    {attribute 'TcHmiSymbol.Show'}
    statuses : M2TiltYAxisStatuses;  (* Statuses of the state machine *)
  END_VAR
  VAR_IN_OUT
    {attribute 'TcHmiSymbol.Show'}
    {attribute 'OPC.UA.DA' := '0'}
    {attribute 'TcHmiSymbol.Hide'}
    config : M2Config;  (* The general M2 config *)
    {attribute 'TcHmiSymbol.Show'}
    {attribute 'OPC.UA.DA' := '0'}
    {attribute 'TcHmiSymbol.Hide'}
    axisConfig : M2PotentiometerAxisConfig;  (* The config particular for this axis *)
  END_VAR

            position(
    config := axisConfig.general.measurement,
    conversionFactor := (constants.POTENTIOMETER_REVOLUTIONS * (constants.SCREW_TO_POT_RATIO * constants.SCREW_PITCH)) / (32768.0 * 1000.0));
statuses.healthStatus(
    isGood := position.statuses.healthStatus.isGood,
    hasWarning := position.statuses.healthStatus.hasWarning);

          

METHOD _log : BOOL
  VAR_INPUT
    {attribute 'TcHmiSymbol.Show'}
    name : STRING;  (* Name of this function block instance *)
  END_VAR
  VAR_IN_OUT
    {attribute 'TcHmiSymbol.Show'}
    buffer : LogBuffer;  (* Buffer to write all logging to *)
  END_VAR
  VAR
    {attribute 'TcHmiSymbol.Show'}
    subBuffer : LogBuffer;  (* Temporary buffer to write logging by parts (sub-statemachines) to *)
  END_VAR
                  LOGGER(
    name := name,
    actualStatus := THIS^.actualStatus,
    previousStatus := THIS^.previousStatus,
    buffer := buffer,
    subBuffer := subBuffer,
    pHealthStatus := ADR(THIS^.statuses.healthStatus));

                
END_METHOD
END_FUNCTION_BLOCK

FUNCTION_BLOCK SM_M2ZAxis
  VAR_INPUT
    {attribute 'TcHmiSymbol.Show'}
    {attribute 'OPC.UA.DA' := '1'}
    {attribute 'OPC.UA.DA.Access' := '1'}
    position : LinearPositionMeasurementU32;  (* Actual position of the axis *)
    {attribute 'TcHmiSymbol.Show'}
    {attribute 'OPC.UA.DA' := '1'}
    {attribute 'OPC.UA.DA.Access' := '1'}
    backlashLifted : BOOL;  (* TRUE if the backlash was previously lifted *)
    {attribute 'TcHmiSymbol.Show'}
    {attribute 'OPC.UA.DA' := '1'}
    {attribute 'OPC.UA.DA.Access' := '1'}
    powered : BOOL;  (* TRUE if the axis is powered *)
    {attribute 'TcHmiSymbol.Show'}
    {attribute 'OPC.UA.DA' := '1'}
    {attribute 'OPC.UA.DA.Access' := '1'}
    isEnabled : BOOL;  (* TRUE if the Z axis control is enabled, FALSE if not *)
  END_VAR
  VAR_OUTPUT
    {attribute 'OPC.UA.DA' := '1'}
    {attribute 'OPC.UA.DA.Access' := '1'}
    {attribute 'TcHmiSymbol.Show'}
    actualStatus : STRING;  (* Current status description *)
    {attribute 'TcHmiSymbol.Show'}
    previousStatus : STRING;  (* Previous status description *)
    {attribute 'TcHmiSymbol.Show'}
    {attribute 'OPC.UA.DA' := '1'}
    {attribute 'OPC.UA.DA.Access' := '1'}
    constants : M2ConstantsZ;  (* Some constants particular for this axis *)
    {attribute 'TcHmiSymbol.Show'}
    statuses : M2ZAxisStatuses;  (* Statuses of the state machine *)
    {attribute 'TcHmiSymbol.Show'}
    parts : M2ZAxisParts;  (* Parts of the state machine *)
  END_VAR
  VAR_IN_OUT
    {attribute 'TcHmiSymbol.Show'}
    {attribute 'OPC.UA.DA' := '0'}
    {attribute 'TcHmiSymbol.Hide'}
    config : M2Config;  (* The general M2 config *)
    {attribute 'TcHmiSymbol.Show'}
    {attribute 'OPC.UA.DA' := '0'}
    {attribute 'TcHmiSymbol.Hide'}
    axisConfig : M2ZAxisConfig;  (* The config particular for this axis *)
  END_VAR

            position(
    rawValue := parts.encoder.counterValue,
    error := parts.encoder.dataError OR (parts.encoder.frameError OR (parts.encoder.powerFailure OR parts.encoder.syncError)),
    config := axisConfig.general.measurement,
    conversionFactor := (constants.SCREW_TO_ENC_RATIO * constants.SCREW_PITCH) / (8192.0 * 1000.0));
parts.highSpeed( isEnabled := isEnabled );
parts.encoder();
statuses.healthStatus(
    isGood := position.statuses.healthStatus.isGood AND parts.encoder.statuses.healthStatus.isGood,
    hasWarning := position.statuses.healthStatus.hasWarning OR parts.encoder.statuses.healthStatus.hasWarning);

          

METHOD _log : BOOL
  VAR_INPUT
    {attribute 'TcHmiSymbol.Show'}
    name : STRING;  (* Name of this function block instance *)
  END_VAR
  VAR_IN_OUT
    {attribute 'TcHmiSymbol.Show'}
    buffer : LogBuffer;  (* Buffer to write all logging to *)
  END_VAR
  VAR
    {attribute 'TcHmiSymbol.Show'}
    subBuffer : LogBuffer;  (* Temporary buffer to write logging by parts (sub-statemachines) to *)
  END_VAR
                  THIS^.parts.highSpeed._log(
    name := 'highSpeed',
    buffer := subBuffer);
THIS^.parts.encoder._log(
    name := 'encoder',
    buffer := subBuffer);
LOGGER(
    name := name,
    actualStatus := THIS^.actualStatus,
    previousStatus := THIS^.previousStatus,
    buffer := buffer,
    subBuffer := subBuffer,
    pHealthStatus := ADR(THIS^.statuses.healthStatus));

                
END_METHOD
END_FUNCTION_BLOCK

FUNCTION_BLOCK SM_M2MoveStepsProcedure
  VAR_INPUT
    {attribute 'TcHmiSymbol.Show'}
    {attribute 'OPC.UA.DA' := '1'}
    {attribute 'OPC.UA.DA.Access' := '1'}
    state : M2MoveProcedureStates;  (* New state, to be set by the manual implementation *)
    {attribute 'TcHmiSymbol.Show'}
    {attribute 'OPC.UA.DA' := '1'}
    {attribute 'OPC.UA.DA.Access' := '1'}
    actualCounterValue AT %I* : UDINT;  (* Actual counter value *)
    {attribute 'TcHmiSymbol.Show'}
    {attribute 'OPC.UA.DA' := '1'}
    {attribute 'OPC.UA.DA.Access' := '1'}
    stepsRemaining : UDINT;  (* Number of steps remaining *)
  END_VAR
  VAR_OUTPUT
    {attribute 'OPC.UA.DA' := '1'}
    {attribute 'OPC.UA.DA.Access' := '1'}
    {attribute 'TcHmiSymbol.Show'}
    actualStatus : STRING;  (* Current status description *)
    {attribute 'TcHmiSymbol.Show'}
    previousStatus : STRING;  (* Previous status description *)
    {attribute 'TcHmiSymbol.Show'}
    statuses : M2MoveStepsProcedureStatuses;  (* Statuses of the state machine *)
  END_VAR
  VAR_IN_OUT
    {attribute 'TcHmiSymbol.Show'}
    {attribute 'OPC.UA.DA' := '0'}
    {attribute 'TcHmiSymbol.Hide'}
    powerOn : Process;
    {attribute 'TcHmiSymbol.Show'}
    {attribute 'OPC.UA.DA' := '0'}
    {attribute 'TcHmiSymbol.Hide'}
    x : M2XAxis;
    {attribute 'TcHmiSymbol.Show'}
    {attribute 'OPC.UA.DA' := '0'}
    {attribute 'TcHmiSymbol.Hide'}
    y : M2YAxis;
    {attribute 'TcHmiSymbol.Show'}
    {attribute 'OPC.UA.DA' := '0'}
    {attribute 'TcHmiSymbol.Hide'}
    z : M2ZAxis;
    {attribute 'TcHmiSymbol.Show'}
    {attribute 'OPC.UA.DA' := '0'}
    {attribute 'TcHmiSymbol.Hide'}
    tiltX : M2TiltXAxis;
    {attribute 'TcHmiSymbol.Show'}
    {attribute 'OPC.UA.DA' := '0'}
    {attribute 'TcHmiSymbol.Hide'}
    tiltY : M2TiltYAxis;
    {attribute 'TcHmiSymbol.Show'}
    {attribute 'OPC.UA.DA' := '0'}
    {attribute 'TcHmiSymbol.Hide'}
    multiplexer : M2Multiplexer;
    {attribute 'TcHmiSymbol.Show'}
    {attribute 'OPC.UA.DA' := '0'}
    {attribute 'TcHmiSymbol.Hide'}
    config : M2Config;
  END_VAR
  VAR
    {attribute 'TcHmiSymbol.Show'}
    {attribute 'OPC.UA.DA' := '1'}
    {attribute 'OPC.UA.DA.Access' := '1'}
    actualCounterValue_ro : UDINT;
  END_VAR

            statuses.busyStatus( isBusy := NOT((state = M2MoveProcedureStates.IDLE) OR ((state = M2MoveProcedureStates.ABORTED) OR (state = M2MoveProcedureStates.ERROR))) );
statuses.healthStatus(
    isGood := NOT(state = M2MoveProcedureStates.ERROR),
    hasWarning := state = M2MoveProcedureStates.ABORTED);
actualCounterValue_ro := actualCounterValue;

          

METHOD _log : BOOL
  VAR_INPUT
    {attribute 'TcHmiSymbol.Show'}
    name : STRING;  (* Name of this function block instance *)
  END_VAR
  VAR_IN_OUT
    {attribute 'TcHmiSymbol.Show'}
    buffer : LogBuffer;  (* Buffer to write all logging to *)
  END_VAR
  VAR
    {attribute 'TcHmiSymbol.Show'}
    subBuffer : LogBuffer;  (* Temporary buffer to write logging by parts (sub-statemachines) to *)
  END_VAR
                  LOGGER(
    name := name,
    actualStatus := THIS^.actualStatus,
    previousStatus := THIS^.previousStatus,
    buffer := buffer,
    subBuffer := subBuffer,
    pHealthStatus := ADR(THIS^.statuses.healthStatus),
    pBusyStatus := ADR(THIS^.statuses.busyStatus));

                
END_METHOD
END_FUNCTION_BLOCK

FUNCTION_BLOCK SM_M2MovePositionProcedure
  VAR_INPUT
    {attribute 'TcHmiSymbol.Show'}
    {attribute 'OPC.UA.DA' := '1'}
    {attribute 'OPC.UA.DA.Access' := '1'}
    state : M2MoveProcedureStates;  (* New state, to be set by the manual implementation *)
  END_VAR
  VAR_OUTPUT
    {attribute 'OPC.UA.DA' := '1'}
    {attribute 'OPC.UA.DA.Access' := '1'}
    {attribute 'TcHmiSymbol.Show'}
    actualStatus : STRING;  (* Current status description *)
    {attribute 'TcHmiSymbol.Show'}
    previousStatus : STRING;  (* Previous status description *)
    {attribute 'TcHmiSymbol.Show'}
    statuses : M2MovePositionProcedureStatuses;  (* Statuses of the state machine *)
  END_VAR
  VAR_IN_OUT
    {attribute 'TcHmiSymbol.Show'}
    {attribute 'OPC.UA.DA' := '0'}
    {attribute 'TcHmiSymbol.Hide'}
    powerOn : Process;
    {attribute 'TcHmiSymbol.Show'}
    {attribute 'OPC.UA.DA' := '0'}
    {attribute 'TcHmiSymbol.Hide'}
    x : M2XAxis;
    {attribute 'TcHmiSymbol.Show'}
    {attribute 'OPC.UA.DA' := '0'}
    {attribute 'TcHmiSymbol.Hide'}
    y : M2YAxis;
    {attribute 'TcHmiSymbol.Show'}
    {attribute 'OPC.UA.DA' := '0'}
    {attribute 'TcHmiSymbol.Hide'}
    z : M2ZAxis;
    {attribute 'TcHmiSymbol.Show'}
    {attribute 'OPC.UA.DA' := '0'}
    {attribute 'TcHmiSymbol.Hide'}
    tiltX : M2TiltXAxis;
    {attribute 'TcHmiSymbol.Show'}
    {attribute 'OPC.UA.DA' := '0'}
    {attribute 'TcHmiSymbol.Hide'}
    tiltY : M2TiltYAxis;
    {attribute 'TcHmiSymbol.Show'}
    {attribute 'OPC.UA.DA' := '0'}
    {attribute 'TcHmiSymbol.Hide'}
    multiplexer : M2Multiplexer;
    {attribute 'TcHmiSymbol.Show'}
    {attribute 'OPC.UA.DA' := '0'}
    {attribute 'TcHmiSymbol.Hide'}
    moveStepsProcedure : M2MoveStepsProcedure;
    {attribute 'TcHmiSymbol.Show'}
    {attribute 'OPC.UA.DA' := '0'}
    {attribute 'TcHmiSymbol.Hide'}
    config : M2Config;
  END_VAR

            statuses.busyStatus( isBusy := NOT((state = M2MoveProcedureStates.IDLE) OR ((state = M2MoveProcedureStates.ABORTED) OR (state = M2MoveProcedureStates.ERROR))) );
statuses.healthStatus(
    isGood := NOT(state = M2MoveProcedureStates.ERROR),
    hasWarning := state = M2MoveProcedureStates.ABORTED);

          

METHOD _log : BOOL
  VAR_INPUT
    {attribute 'TcHmiSymbol.Show'}
    name : STRING;  (* Name of this function block instance *)
  END_VAR
  VAR_IN_OUT
    {attribute 'TcHmiSymbol.Show'}
    buffer : LogBuffer;  (* Buffer to write all logging to *)
  END_VAR
  VAR
    {attribute 'TcHmiSymbol.Show'}
    subBuffer : LogBuffer;  (* Temporary buffer to write logging by parts (sub-statemachines) to *)
  END_VAR
                  LOGGER(
    name := name,
    actualStatus := THIS^.actualStatus,
    previousStatus := THIS^.previousStatus,
    buffer := buffer,
    subBuffer := subBuffer,
    pHealthStatus := ADR(THIS^.statuses.healthStatus),
    pBusyStatus := ADR(THIS^.statuses.busyStatus));

                
END_METHOD
END_FUNCTION_BLOCK

FUNCTION_BLOCK M2SelectAxisProcess EXTENDS BaseProcess
  VAR_INPUT
    {attribute 'OPC.UA.DA' := '1'}
    {attribute 'TcHmiSymbol.Show'}
    set : M2SelectAxisProcessArgs;  (* Arguments to be set, before writing do_request TRUE *)
  END_VAR
  VAR_OUTPUT
    {attribute 'OPC.UA.DA' := '1'}
    {attribute 'OPC.UA.DA.Access' := '1'}
    {attribute 'TcHmiSymbol.Show'}
    get : M2SelectAxisProcessArgs;  (* Arguments in use by the process, if do_request was accepted *)
  END_VAR

            IF do_request THEN
    do_request_result := request( axis := set.axis );
    do_request := FALSE;
END_IF;
SUPER^();

          

{attribute 'TcRpcEnable' := '1'}
METHOD start
  VAR_INPUT
    {attribute 'TcHmiSymbol.Show'}
    axis : M2Axes;  (* The axis to select *)
  END_VAR
                  THIS^.get.axis := axis;
THIS^.statuses.busyStatus( isBusy := TRUE );
THIS^.statuses.healthStatus( isGood := TRUE );

                
END_METHOD

{attribute 'TcRpcEnable' := '1'}
METHOD request : RequestResults
  VAR_INPUT
    {attribute 'TcHmiSymbol.Show'}
    axis : M2Axes;  (* The axis to select *)
  END_VAR
                  IF THIS^.statuses.enabledStatus.enabled THEN
    request := RequestResults.ACCEPTED;
    THIS^.start( axis := axis );
ELSE
    request := RequestResults.REJECTED;
END_IF;

                
END_METHOD
END_FUNCTION_BLOCK

FUNCTION_BLOCK M2MoveProcess EXTENDS BaseProcess
  VAR_INPUT
    {attribute 'OPC.UA.DA' := '1'}
    {attribute 'TcHmiSymbol.Show'}
    set : M2MoveProcessArgs;  (* Arguments to be set, before writing do_request TRUE *)
  END_VAR
  VAR_OUTPUT
    {attribute 'OPC.UA.DA' := '1'}
    {attribute 'OPC.UA.DA.Access' := '1'}
    {attribute 'TcHmiSymbol.Show'}
    get : M2MoveProcessArgs;  (* Arguments in use by the process, if do_request was accepted *)
  END_VAR

            IF do_request THEN
    do_request_result := request(
    axis := set.axis,
    position := set.position);
    do_request := FALSE;
END_IF;
SUPER^();

          

{attribute 'TcRpcEnable' := '1'}
METHOD start
  VAR_INPUT
    {attribute 'TcHmiSymbol.Show'}
    axis : M2Axes;  (* The axis to move *)
    {attribute 'TcHmiSymbol.Show'}
    position : LREAL;  (* Move to a certain position in millimeters *)
  END_VAR
                  THIS^.get.axis := axis;
THIS^.get.position := position;
THIS^.statuses.busyStatus( isBusy := TRUE );
THIS^.statuses.healthStatus( isGood := TRUE );

                
END_METHOD

{attribute 'TcRpcEnable' := '1'}
METHOD request : RequestResults
  VAR_INPUT
    {attribute 'TcHmiSymbol.Show'}
    axis : M2Axes;  (* The axis to move *)
    {attribute 'TcHmiSymbol.Show'}
    position : LREAL;  (* Move to a certain position in millimeters *)
  END_VAR
                  IF THIS^.statuses.enabledStatus.enabled THEN
    request := RequestResults.ACCEPTED;
    THIS^.start(
        axis := axis,
        position := position);
ELSE
    request := RequestResults.REJECTED;
END_IF;

                
END_METHOD
END_FUNCTION_BLOCK

FUNCTION_BLOCK M2MoveStepsProcess EXTENDS BaseProcess
  VAR_INPUT
    {attribute 'OPC.UA.DA' := '1'}
    {attribute 'TcHmiSymbol.Show'}
    set : M2MoveStepsProcessArgs;  (* Arguments to be set, before writing do_request TRUE *)
  END_VAR
  VAR_OUTPUT
    {attribute 'OPC.UA.DA' := '1'}
    {attribute 'OPC.UA.DA.Access' := '1'}
    {attribute 'TcHmiSymbol.Show'}
    get : M2MoveStepsProcessArgs;  (* Arguments in use by the process, if do_request was accepted *)
  END_VAR

            IF do_request THEN
    do_request_result := request(
    axis := set.axis,
    steps := set.steps,
    cw := set.cw,
    fast := set.fast);
    do_request := FALSE;
END_IF;
SUPER^();

          

{attribute 'TcRpcEnable' := '1'}
METHOD start
  VAR_INPUT
    {attribute 'TcHmiSymbol.Show'}
    axis : M2Axes;  (* The axis to move *)
    {attribute 'TcHmiSymbol.Show'}
    steps : UDINT;  (* Move a certain number of steps *)
    {attribute 'TcHmiSymbol.Show'}
    cw : BOOL;  (* True if the axis should be moved in CW (negative) direction *)
    {attribute 'TcHmiSymbol.Show'}
    fast : BOOL;  (* True if the axis should be moved fast (only used in case of Z-axis!) *)
  END_VAR
                  THIS^.get.axis := axis;
THIS^.get.steps := steps;
THIS^.get.cw := cw;
THIS^.get.fast := fast;
THIS^.statuses.busyStatus( isBusy := TRUE );
THIS^.statuses.healthStatus( isGood := TRUE );

                
END_METHOD

{attribute 'TcRpcEnable' := '1'}
METHOD request : RequestResults
  VAR_INPUT
    {attribute 'TcHmiSymbol.Show'}
    axis : M2Axes;  (* The axis to move *)
    {attribute 'TcHmiSymbol.Show'}
    steps : UDINT;  (* Move a certain number of steps *)
    {attribute 'TcHmiSymbol.Show'}
    cw : BOOL;  (* True if the axis should be moved in CW (negative) direction *)
    {attribute 'TcHmiSymbol.Show'}
    fast : BOOL;  (* True if the axis should be moved fast (only used in case of Z-axis!) *)
  END_VAR
                  IF THIS^.statuses.enabledStatus.enabled THEN
    request := RequestResults.ACCEPTED;
    THIS^.start(
        axis := axis,
        steps := steps,
        cw := cw,
        fast := fast);
ELSE
    request := RequestResults.REJECTED;
END_IF;

                
END_METHOD
END_FUNCTION_BLOCK

FUNCTION_BLOCK M2DoThermalFocusForStationPosition EXTENDS BaseProcess
  VAR_INPUT
    {attribute 'OPC.UA.DA' := '1'}
    {attribute 'TcHmiSymbol.Show'}
    set : M2DoThermalFocusForStationPositionArgs;  (* Arguments to be set, before writing do_request TRUE *)
  END_VAR
  VAR_OUTPUT
    {attribute 'OPC.UA.DA' := '1'}
    {attribute 'OPC.UA.DA.Access' := '1'}
    {attribute 'TcHmiSymbol.Show'}
    get : M2DoThermalFocusForStationPositionArgs;  (* Arguments in use by the process, if do_request was accepted *)
  END_VAR

            IF do_request THEN
    do_request_result := request( station := set.station );
    do_request := FALSE;
END_IF;
SUPER^();

          

{attribute 'TcRpcEnable' := '1'}
METHOD start
  VAR_INPUT
    {attribute 'TcHmiSymbol.Show'}
    station : M3PositionIDs;  (* The station numerical ID for which the thermal focus should be executed *)
  END_VAR
                  THIS^.get.station := station;
THIS^.statuses.busyStatus( isBusy := TRUE );
THIS^.statuses.healthStatus( isGood := TRUE );

                
END_METHOD

{attribute 'TcRpcEnable' := '1'}
METHOD request : RequestResults
  VAR_INPUT
    {attribute 'TcHmiSymbol.Show'}
    station : M3PositionIDs;  (* The station numerical ID for which the thermal focus should be executed *)
  END_VAR
                  IF THIS^.statuses.enabledStatus.enabled THEN
    request := RequestResults.ACCEPTED;
    THIS^.start( station := station );
ELSE
    request := RequestResults.REJECTED;
END_IF;

                
END_METHOD
END_FUNCTION_BLOCK

FUNCTION_BLOCK M2DoThermalFocusForStationName EXTENDS BaseProcess
  VAR_INPUT
    {attribute 'OPC.UA.DA' := '1'}
    {attribute 'TcHmiSymbol.Show'}
    set : M2DoThermalFocusForStationNameArgs;  (* Arguments to be set, before writing do_request TRUE *)
  END_VAR
  VAR_OUTPUT
    {attribute 'OPC.UA.DA' := '1'}
    {attribute 'OPC.UA.DA.Access' := '1'}
    {attribute 'TcHmiSymbol.Show'}
    get : M2DoThermalFocusForStationNameArgs;  (* Arguments in use by the process, if do_request was accepted *)
  END_VAR

            IF do_request THEN
    do_request_result := request( station := set.station );
    do_request := FALSE;
END_IF;
SUPER^();

          

{attribute 'TcRpcEnable' := '1'}
METHOD start
  VAR_INPUT
    {attribute 'TcHmiSymbol.Show'}
    station : STRING;  (* The configured station name, for which the thermal focus should be executed *)
  END_VAR
                  THIS^.get.station := station;
THIS^.statuses.busyStatus( isBusy := TRUE );
THIS^.statuses.healthStatus( isGood := TRUE );

                
END_METHOD

{attribute 'TcRpcEnable' := '1'}
METHOD request : RequestResults
  VAR_INPUT
    {attribute 'TcHmiSymbol.Show'}
    station : STRING;  (* The configured station name, for which the thermal focus should be executed *)
  END_VAR
                  IF THIS^.statuses.enabledStatus.enabled THEN
    request := RequestResults.ACCEPTED;
    THIS^.start( station := station );
ELSE
    request := RequestResults.REJECTED;
END_IF;

                
END_METHOD
END_FUNCTION_BLOCK
